TYPE JSON_Drive :
	STRUCT
		  id 		: DINT;
		  name 		: STRING(255);
		  speed 	: LREAL;
		  torquerel : LREAL;
		  torque	: LREAL;
	END_STRUCT
END_TYPE

(* stored: Version 1.1.0.1
   DUT JSON_Drive: Id {30f2acbf-f420-0594-1614-25c7c85318f3} *)
